PROGRAM pouS4Alarms
VAR
	idbMsgAlarm: FB_CheckMessageBounds;

END_VAR

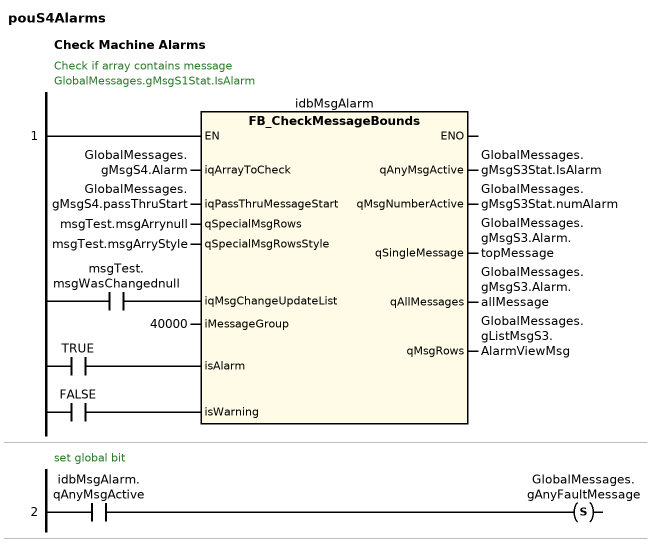
// NETWORK 1: Check Machine Alarms
// Check if array contains message
//
// GlobalMessages.gMsgS1Stat.IsAlarm
idbMsgAlarm(
    iqArrayToCheck := GlobalMessages.gMsgS4.Alarm,
    iqPassThruMessageStart := GlobalMessages.gMsgS4.passThruStart,
    qSpecialMsgRows := msgTest.msgArrynull,
    qSpecialMsgRowsStyle := msgTest.msgArryStyle,
    iqMsgChangeUpdateList := msgTest.msgWasChangednull,
    iMessageGroup := 40000,
    isAlarm := TRUE,
    isWarning := FALSE,
    qAnyMsgActive => GlobalMessages.gMsgS3Stat.IsAlarm,
    qMsgNumberActive => GlobalMessages.gMsgS3Stat.numAlarm,
    qSingleMessage => GlobalMessages.gMsgS3.Alarm.topMessage,
    qAllMessages => GlobalMessages.gMsgS3.Alarm.allMessage,
    qMsgRows => GlobalMessages.gListMsgS3.AlarmViewMsg); // FB_CheckMessageBounds

// NETWORK 2
// set global bit
GlobalMessages.gAnyFaultMessage S= idbMsgAlarm.qAnyMsgActive;

END_PROGRAM

(* stored: Version 1.1.0.1, ProductVersion 3.1.4024.12
   POU pouS4Alarms: Id {c4aa73c4-1839-47a1-a4ef-867737da48c3}, SpecialFunc None *)
